(*
SPDX-FileCopyrightText: Â© 2026 Oleksandr Tiutyk <trofimich@gmail.com>
SPDX-License-Identifier: MIT
License: https://opensource.org/license/mit
*)

(*!
<summary>Provides automation component operational state and diagnostics to an HMI.</summary>
<description>
Aggregates enablement, error details, and current operational state information for UI visualization.
</description>
*)

TYPE HMI_AUTOMATION_COMPONENT_STATUSES :
STRUCT
	Enabled : BOOL;

	HasError : BOOL;
	ErrorMessage : TOF_Core.ERROR_MESSAGE;
	ErrorSource : STRING(255);
	ErrorLocalTimestamp : LDATE_AND_TIME;
	ErrorUtcTimestamp : LDATE_AND_TIME;

	OperationalState : OPERATIONAL_STATE;
	OperationalStateName : STRING;
	OperationalStateReason : WSTRING(255);
END_STRUCT
END_TYPE

(* stored: Version 1.1.0.1
   DUT HMI_AUTOMATION_COMPONENT_STATUSES: Id {c40c7e9a-c43b-4973-93e1-8c17864d5829} *)
